{attribute 'OPC.UA.DA' := '0'}
TYPE RFactorSettings EXTENDS RFactorBase :
STRUCT
END_STRUCT
END_TYPE

(* stored: Version 1.1.0.1, ProductVersion 3.1.4024.4
   DUT RFactorSettings: Id {fb1bb082-ef22-4e85-a845-75f7adc62ccb} *)
